{attribute 'linkalways'} 
{attribute 'no_explicit_call' := 'This FB is a CLASS and must be accessed using methods or properties'}
{attribute 'enable_dynamic_creation'}
FUNCTION_BLOCK Node_F_VN_SetAt_TcVnVector2_SINT EXTENDS VisionNode
VAR
    aElement : _TcVnVector2_SINT;
    ipContainer : _ITcVnContainer;
    nIndex : _ULINT(0);
    hrPrev : _HRESULT(S_OK);
    hresult : _HRESULT(S_OK);
END_VAR

METHOD PUBLIC  Clone : I_Node
VAR
	pNode : POINTER TO Node_F_VN_SetAt_TcVnVector2_SINT;
END_VAR
pNode := __NEW(Node_F_VN_SetAt_TcVnVector2_SINT);
Clone := pNode^;
END_METHOD

METHOD FB_init : BOOL
VAR_INPUT
	bInitRetains : BOOL; // if TRUE, the retain variables are initialized (warm start / cold start)
	bInCopyCode : BOOL;  // if TRUE, the instance afterwards gets moved into the copy code (online change)
END_VAR
AddInput('aElement', aElement);
AddInput('ipContainer', ipContainer);
AddInput('nIndex', nIndex);
AddInput('hrPrev', hrPrev);
AddOutput('ipContainer', ipContainer);
AddOutput('hresult',hresult);
END_METHOD

METHOD PROTECTED OnExecute : HRESULT
hresult.Value := F_VN_SetAt_TcVnVector2_SINT(
    aElement := aElement.Value,
    ipContainer := ipContainer.Value,
    nIndex := nIndex.Value,
    hrPrev:= hrPrev.Value);
END_METHOD

METHOD PUBLIC PreExecutionCheck
VAR_INPUT
	Check : I_PreExecutionChecks;
END_VAR
Check.IsTrue(ipContainer.IsValid, 'ipContainer must be a valid container');
END_METHOD

END_FUNCTION_BLOCK

(* stored: Version 1.1.0.1, ProductVersion 3.1.4024.13
   POU Node_F_VN_SetAt_TcVnVector2_SINT: Id {6b9b296d-2b5e-40fe-8071-8dc096851f51}, SpecialFunc None
   Folder Constructor: Id {6fff0a6b-2408-4e15-af28-81750b169637}
   Method Clone: Id {50f2813e-9877-423f-9e7e-fd3a3a005655}
   Method FB_init: Id {6948fa12-add0-4a91-abf6-415fe85e3ea0}
   Method OnExecute: Id {88e828f4-6895-48a6-b9cd-cba29a910b02}
   Method PreExecutionCheck: Id {cf2a88d6-b942-40d3-a809-6c83dea13b4c} *)
